FUNCTION_BLOCK DummyRollgang (* Demonstrate self initialize with data from an XML database by Xquery *)
  (* Standard: 61499-2; Description: Copyright (c) 2025 Monika Wenger This program and the accompanying materials are made available under the terms of the Eclipse Public License 2.0 which is available at https://www.eclipse.org/legal/epl-2.0/ SPDX-License-Identifier: EPL-2.0 *)
  (* Version 1.0, 2025-05-18, Monika Wenger *)
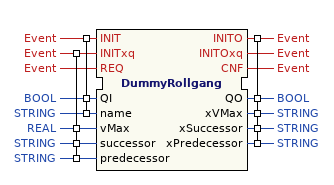
  EVENT_INPUT
    INIT WITH QI, name; (* Initialization Request *)
    INITxq WITH vMax, successor, predecessor;
    REQ; (* Normal Execution Request *)
  END_EVENT
  EVENT_OUTPUT
    INITO WITH QO, xVMax, xSuccessor, xPredecessor; (* Initialization Confirm *)
    INITOxq;
    CNF; (* Execution Confirmation *)
  END_EVENT
  VAR_INPUT
    QI : BOOL; (* Input event qualifier *)
    name : STRING; (* name of this Rollgang *)
    vMax : REAL; (* maximal velocity *)
    successor : STRING; (* name of the successor Rollgang *)
    predecessor : STRING; (* name of the predecessor Rollgang *)
  END_VAR
  VAR_OUTPUT
    QO : BOOL; (* Output event qualifier *)
    xVMax : STRING; (* Xquery to get maximal velocity *)
    xSuccessor : STRING; (* Xquery to get name of the successor Rollgang *)
    xPredecessor : STRING; (* Xquery to get name of the predecessor Rollgang *)
  END_VAR
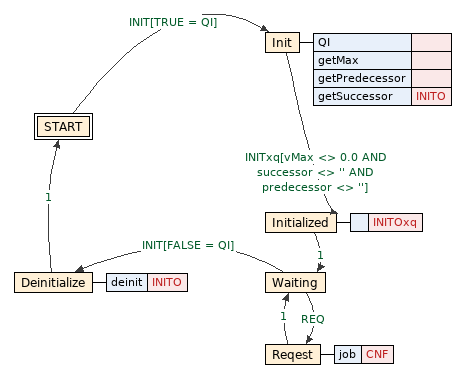
  EC_STATES
    START; (* Initial State *)
    Init : QI, getMax, getPredecessor, getSuccessor -> INITO; (* Initialization *)
    Initialized : -> INITOxq;
    Reqest : job -> CNF;
    Waiting;
    Deinitialize : deinit -> INITO;
  END_STATES
  EC_TRANSITIONS
    START TO Init := INIT[TRUE = QI];
    Init TO Initialized := INITxq[vMax <> 0.0 AND successor <> '' AND predecessor <> ''];
    Initialized TO Waiting := 1;
    Waiting TO Reqest := REQ;
    Reqest TO Waiting := 1;
    Waiting TO Deinitialize := INIT[FALSE = QI];
    Deinitialize TO START := 1;
  END_TRANSITIONS
  ALGORITHM QI IN ST:
QO := QI;
  END_ALGORITHM
  ALGORITHM deinit IN ST:
QO := FALSE;
  END_ALGORITHM
  ALGORITHM getMax IN ST:
xVMax := CONCAT('xquery ', STRING#'let $$name := $'', name, STRING#'$' ',
	'let $$component := //InstanceHierarchy/*/InternalElement[@Name=$$name] ',
	'let $$compType := tokenize($$component/RoleRequirements/@RefBaseRoleClassPath/data(),$'/$')[last()] ',
	'let $$rollerTable :=  $$component/InternalElement/RoleRequirements[contains(@RefBaseRoleClassPath,$'RollConveyor$')]/.. ',
	'let $$rollDiameter := $$rollerTable/Attribute[@Name=$'RollDiameter$']/Value/data() ',
	'let $$link := tokenize($$component/InternalLink/@RefPartnerSideA/data(),$':$')[1] ',
	'let $$motor := //InternalElement[@ID=$$link]/RoleRequirements[contains(@RefBaseRoleClassPath,$'ElectricMotor$')]/.. ',
	'let $$gearFactor := $$motor/Attribute[@Name=$'Gearfactor$']/Value/data() ',
	'let $$rotSpeed := $$motor/Attribute[@Name=$'Rotational Speed$']/Value/data() ',
	STRING#'let $$linSpeed :=  $$rotSpeed div (60.0 * $$gearFactor) * (2.0 * 3.1416 * 0.5 * $$rollDiameter) ',
	STRING#'return round-half-to-even($$linSpeed, 3)');
  END_ALGORITHM
  ALGORITHM getPredecessor IN ST:
xPredecessor := CONCAT(STRING#'xquery ', STRING#'let $$name := $'', name, STRING#'$' ',
	STRING#'let $$links := //InstanceHierarchy/InternalElement/InternalLink ',
	STRING#'let $$cp := //InstanceHierarchy/*/InternalElement[@Name=$$name] ', STRING#'let $$id := $$cp/@ID/data() ',
	STRING#'let $$succId := tokenize($$links[contains(@RefPartnerSideB, $$id)]/@RefPartnerSideA, $':$')[1] ',
	STRING#'let $$successor := //InstanceHierarchy/*/InternalElement[@ID=$$succId] ',
	STRING# 'return $$successor/@Name/data() ');
  END_ALGORITHM
  ALGORITHM getSuccessor IN ST:
xSuccessor := CONCAT('xquery ', STRING#'let $$name := $'', name, STRING#'$' ',
	STRING#'let $$links := //InstanceHierarchy/InternalElement/InternalLink ',
	STRING#'let $$cp := //InstanceHierarchy/*/InternalElement[@Name=$$name] ', STRING#'let $$id := $$cp/@ID/data() ',
	STRING#'let $$succId := tokenize($$links[contains(@RefPartnerSideA, $$id)]/@RefPartnerSideB, $':$')[1] ',
	STRING#'let $$successor := //InstanceHierarchy/*/InternalElement[@ID=$$succId] ',
	STRING# 'return $$successor/@Name/data() ');
  END_ALGORITHM
  ALGORITHM job IN ST:
// do my job
  END_ALGORITHM
END_FUNCTION_BLOCK
